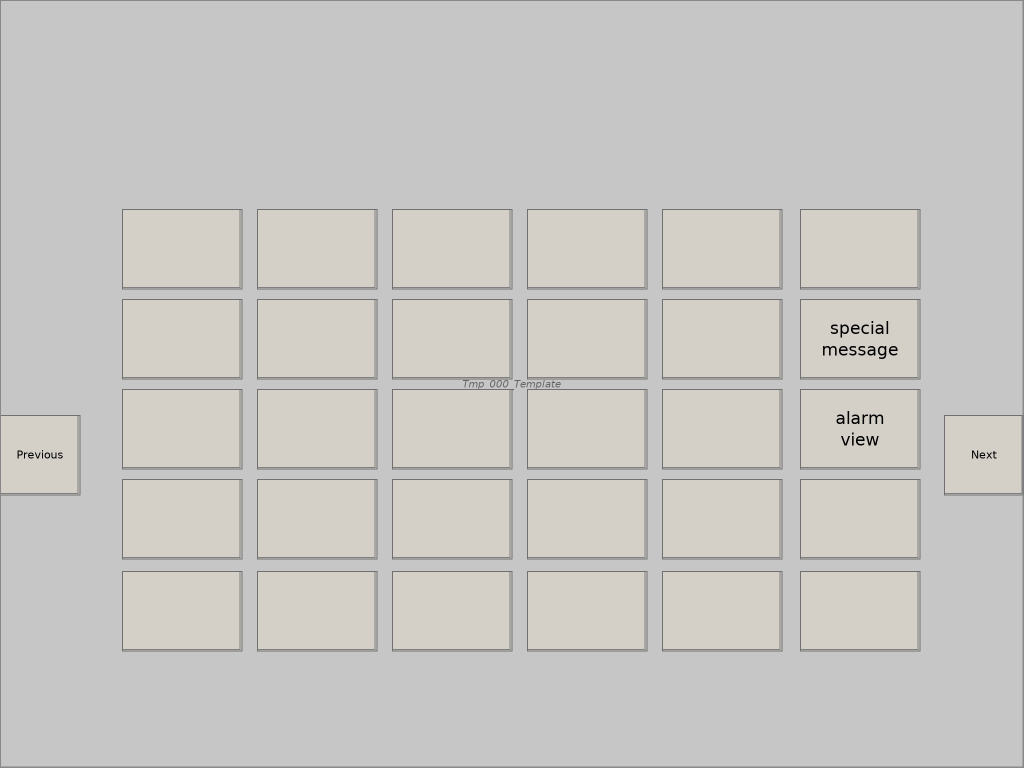
VISUALIZATION Men_032_MenuScreen_3  // 1024x768
    Frame (0,0 1024x768)
        shows Tmp_000_Template(header := gHMIData.hmiHeader)
    Group (0,415 1024x80)
        Button (0,0 80x80), "Previous"
            OnMouseClick: change screen: Men_031_MenuScreen_2
            OnMouseDown: execute { gHMIButtons.gAnyButtonPressed := TRUE; }
        Button (944,0 80x80), "Next"
            OnMouseClick: change screen: Men_030_MenuScreen
            OnMouseDown: execute { gHMIButtons.gAnyButtonPressed := TRUE; }
    Button (800,299 120x80), "special message", text list: ''
        OnMouseClick: change screen: Msg_020_Alarms
        OnMouseDown: execute { gHMIButtons.gAnyButtonPressed := TRUE; }
    Button (800,389 120x80), "alarm view", text list: ''
        OnMouseClick: change screen: Msg_021_AlarmsView
        OnMouseDown: execute { gHMIButtons.gAnyButtonPressed := TRUE; }
    Button (122,209 120x80), text list: ''
        OnMouseDown: execute { gHMIButtons.gAnyButtonPressed := TRUE; }
    Button (257,209 120x80), text list: ''
        OnMouseDown: execute { gHMIButtons.gAnyButtonPressed := TRUE; }
    Button (392,209 120x80), text list: ''
        OnMouseDown: execute { gHMIButtons.gAnyButtonPressed := TRUE; }
    Button (527,209 120x80), text list: ''
        OnMouseDown: execute { gHMIButtons.gAnyButtonPressed := TRUE; }
    Button (662,209 120x80), text list: ''
        OnMouseDown: execute { gHMIButtons.gAnyButtonPressed := TRUE; }
    Button (800,209 120x80), text list: ''
        OnMouseDown: execute { gHMIButtons.gAnyButtonPressed := TRUE; }
    Button (122,299 120x80), text list: ''
        OnMouseDown: execute { gHMIButtons.gAnyButtonPressed := TRUE; }
    Button (257,299 120x80), text list: ''
        OnMouseDown: execute { gHMIButtons.gAnyButtonPressed := TRUE; }
    Button (392,299 120x80), text list: ''
        OnMouseDown: execute { gHMIButtons.gAnyButtonPressed := TRUE; }
    Button (527,299 120x80), text list: ''
        OnMouseDown: execute { gHMIButtons.gAnyButtonPressed := TRUE; }
    Button (662,299 120x80), text list: ''
        OnMouseDown: execute { gHMIButtons.gAnyButtonPressed := TRUE; }
    Button (122,389 120x80), text list: ''
        OnMouseDown: execute { gHMIButtons.gAnyButtonPressed := TRUE; }
    Button (257,389 120x80), text list: ''
        OnMouseDown: execute { gHMIButtons.gAnyButtonPressed := TRUE; }
    Button (392,389 120x80), text list: ''
        OnMouseDown: execute { gHMIButtons.gAnyButtonPressed := TRUE; }
    Button (527,389 120x80), text list: ''
        OnMouseDown: execute { gHMIButtons.gAnyButtonPressed := TRUE; }
    Button (662,389 120x80), text list: ''
        OnMouseDown: execute { gHMIButtons.gAnyButtonPressed := TRUE; }
    Button (122,479 120x80), text list: ''
        OnMouseDown: execute { gHMIButtons.gAnyButtonPressed := TRUE; }
    Button (257,479 120x80), text list: ''
        OnMouseDown: execute { gHMIButtons.gAnyButtonPressed := TRUE; }
    Button (392,479 120x80), text list: ''
        OnMouseDown: execute { gHMIButtons.gAnyButtonPressed := TRUE; }
    Button (527,479 120x80), text list: ''
        OnMouseDown: execute { gHMIButtons.gAnyButtonPressed := TRUE; }
    Button (662,479 120x80), text list: ''
        OnMouseDown: execute { gHMIButtons.gAnyButtonPressed := TRUE; }
    Button (800,479 120x80), text list: ''
        OnMouseDown: execute { gHMIButtons.gAnyButtonPressed := TRUE; }
    Button (122,571 120x80), text list: ''
        OnMouseDown: execute { gHMIButtons.gAnyButtonPressed := TRUE; }
    Button (257,571 120x80), text list: ''
        OnMouseDown: execute { gHMIButtons.gAnyButtonPressed := TRUE; }
    Button (392,571 120x80), text list: ''
        OnMouseDown: execute { gHMIButtons.gAnyButtonPressed := TRUE; }
    Button (527,571 120x80), text list: ''
        OnMouseDown: execute { gHMIButtons.gAnyButtonPressed := TRUE; }
    Button (662,571 120x80), text list: ''
        OnMouseDown: execute { gHMIButtons.gAnyButtonPressed := TRUE; }
    Button (800,571 120x80), text list: ''
        OnMouseDown: execute { gHMIButtons.gAnyButtonPressed := TRUE; }
END_VISUALIZATION

(* stored: Version 1.1.0.1, ProductVersion 3.1.4024.11
   Visu Men_032_MenuScreen_3: Id {73b9ea03-2c91-46d6-a0f2-36ef36d02055} *)
